// Create errors with specified parameters and sets the timestamp to the local time from a starting range.
// Some error descriptors have ranges for error codes.
// If the code is 0 an unraised error is created.
FUNCTION F_CreateErrorFromStartRange : T_Error // Instance of created error.
VAR_INPUT
	ipDescriptor 	: I_ErrorDescriptor; 	// Error descriptor.
	StartRange		: T_ErrorCode;			// Error code starting Range. 
	Code 			: T_ErrorCode; 			// Error code.
END_VAR
VAR
	fbMutError 			: FB_MutableError;
	nResult,
	nLowResTimestamp 	: DWORD;
	nHighResTimestamp 	: ULINT;
END_VAR

// Get high res. local timestamp.
nResult := SysTimeRtc.SysTimeRtcConvertUtcToLocal(
			SysTimeRtc.SysTimeRtcGet(nResult),
			nLowResTimestamp);

// Add milliseconds to high res. timestamp.
nHighResTimestamp := TO_ULINT(nLowResTimestamp)*1000 
					 + 
					 (TO_ULINT(LTIME()) MOD TO_ULINT(LTIME#1S)) / TO_ULINT(LTIME#1MS);

// Set muttable error.
fbMutError.SetDescriptor(ipDescriptor)
		  .RaiseError(SEL(Code <> 0, 0, StartRange + Code))
		  .SetTimestamp(nHighResTimestamp);
		  
// Return as immutable error.
F_CreateErrorFromStartRange := fbMutError;

END_FUNCTION

(* stored: Version 1.1.0.1
   POU F_CreateErrorFromStartRange: Id {d5f028a0-24ee-0f73-1be1-cd20ce46f9c4}, SpecialFunc None *)
